PROGRAM PRG_CNCVariablesViewer
VAR			
	fbReadCNCVariables : FB_ReadCNCVariables;		
END_VAR

fbReadCNCVariables(
	bEnable:= TRUE, 
	nChanIdx:= PLCSelectedChannel, 
	eVariablesType:= eVariablesType, 
	tIntervall:= T#1S, 	 
	stCNCVariablesViewer_Data:= stCNCVariablesViewer_Data);

END_PROGRAM

(* stored: Version 1.1.0.1, ProductVersion 3.1.4022.6
   POU PRG_CNCVariablesViewer: Id {da8e67fd-e008-4579-a9d5-34610f25362d}, SpecialFunc None *)
